{attribute 'qualified_only'}
VAR_GLOBAL
	bProjectA : BOOL := FALSE;
END_VAR

(* stored: Version 1.1.0.1, ProductVersion 3.1.4022.18
   GVL GVL_ProjectA: Id {673572d4-45ac-407d-b34c-97a1056b4dba} *)
